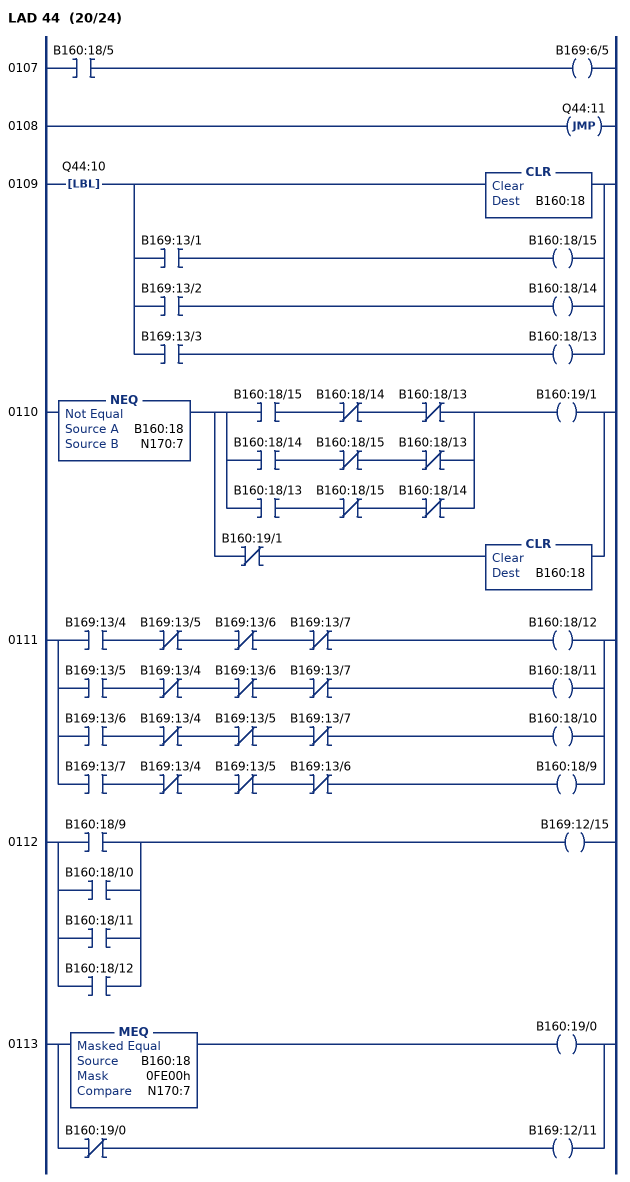
% Rung: 107 %
SOR XIC B160:18/5 OTE B169:6/5 EOR
% Rung: 108 %
SOR JMP Q44:11 EOR
% Rung: 109 %
SOR LBL Q44:10 BST CLR B160:18 NXB XIC B169:13/1 OTE B160:18/15 NXB XIC B169:13/2 OTE B160:18/14 NXB XIC B169:13/3 OTE B160:18/13 BND EOR
% Rung: 110 %
SOR NEQ B160:18 N170:7 BST BST XIC B160:18/15 XIO B160:18/14 XIO B160:18/13 NXB XIC B160:18/14 XIO B160:18/15 XIO B160:18/13 NXB XIC B160:18/13 XIO B160:18/15 XIO B160:18/14 BND OTE B160:19/1 NXB XIO B160:19/1 CLR B160:18 BND EOR
% Rung: 111 %
SOR BST XIC B169:13/4 XIO B169:13/5 XIO B169:13/6 XIO B169:13/7 OTE B160:18/12 NXB XIC B169:13/5 XIO B169:13/4 XIO B169:13/6 XIO B169:13/7 OTE B160:18/11 NXB XIC B169:13/6 XIO B169:13/4 XIO B169:13/5 XIO B169:13/7 OTE B160:18/10 NXB XIC B169:13/7 XIO B169:13/4 XIO B169:13/5 XIO B169:13/6 OTE B160:18/9 BND EOR
% Rung: 112 %
SOR BST XIC B160:18/9 NXB XIC B160:18/10 NXB XIC B160:18/11 NXB XIC B160:18/12 BND OTE B169:12/15 EOR
% Rung: 113 %
SOR BST MEQ B160:18 0FE00h N170:7 OTE B160:19/0 NXB XIO B160:19/0 OTE B169:12/11 BND EOR

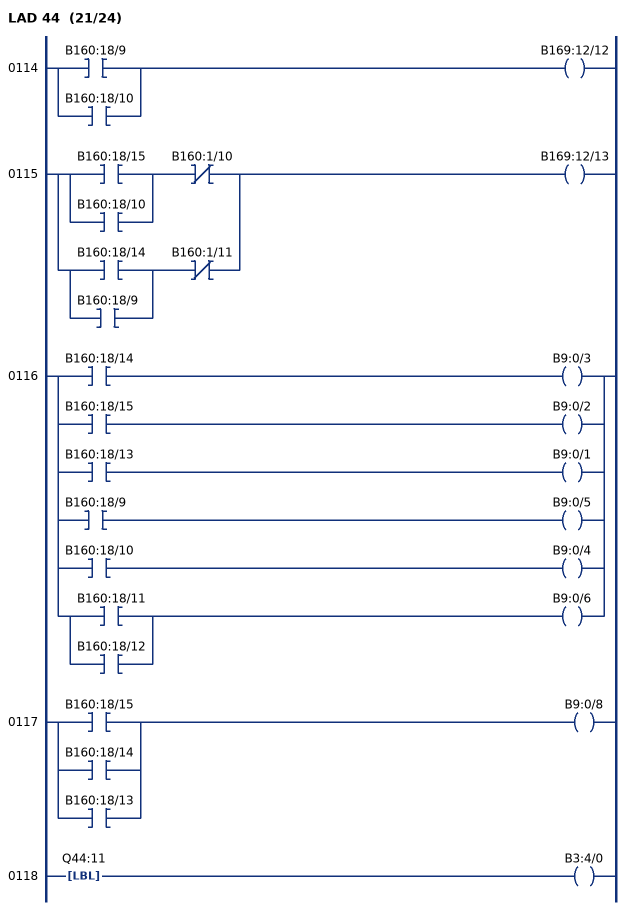
% Rung: 114 %
SOR BST XIC B160:18/9 NXB XIC B160:18/10 BND OTE B169:12/12 EOR
% Rung: 115 %
SOR BST BST XIC B160:18/15 NXB XIC B160:18/10 BND XIO B160:1/10 NXB BST XIC B160:18/14 NXB XIC B160:18/9 BND XIO B160:1/11 BND OTE B169:12/13 EOR
% Rung: 116 %
SOR BST XIC B160:18/14 OTE B9:0/3 NXB XIC B160:18/15 OTE B9:0/2 NXB XIC B160:18/13 OTE B9:0/1 NXB XIC B160:18/9 OTE B9:0/5 NXB XIC B160:18/10 OTE B9:0/4 NXB BST XIC B160:18/11 NXB XIC B160:18/12 BND OTE B9:0/6 BND EOR
% Rung: 117 %
SOR BST XIC B160:18/15 NXB XIC B160:18/14 NXB XIC B160:18/13 BND OTE B9:0/8 EOR
% Rung: 118 %
SOR LBL Q44:11 OTE B3:4/0 EOR

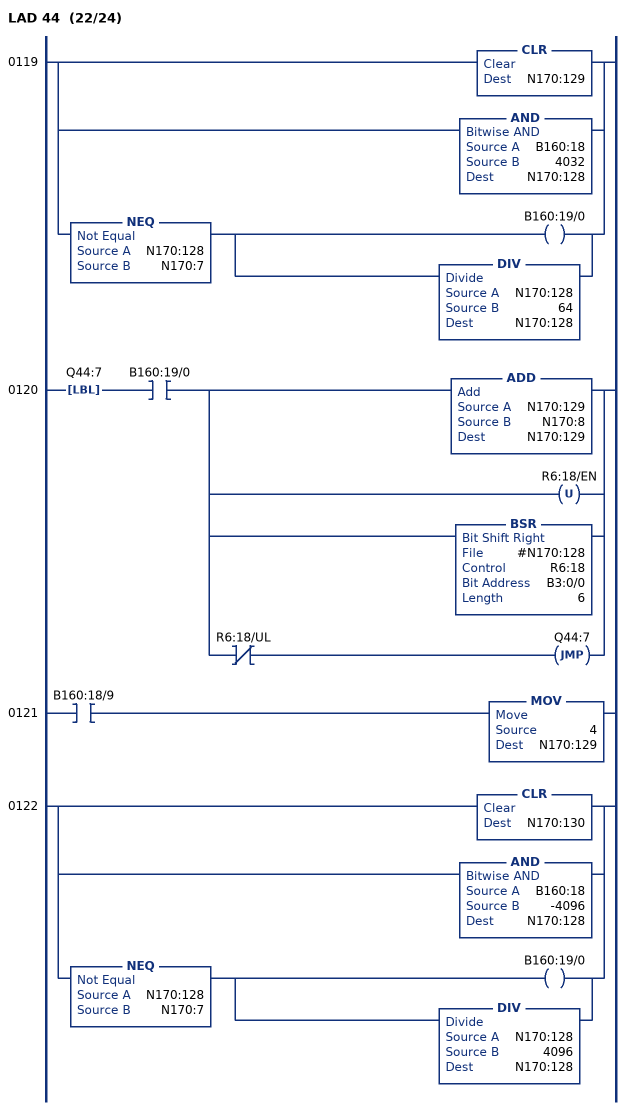
% Rung: 119 %
SOR BST CLR N170:129 NXB AND B160:18 4032 N170:128 NXB NEQ N170:128 N170:7 BST OTE B160:19/0 NXB DIV N170:128 64 N170:128 BND BND EOR
% Rung: 120 %
SOR LBL Q44:7 XIC B160:19/0 BST ADD N170:129 N170:8 N170:129 NXB OTU R6:18/EN NXB BSR #N170:128 R6:18 B3:0/0 6 NXB XIO R6:18/UL JMP Q44:7 BND EOR
% Rung: 121 %
SOR XIC B160:18/9 MOV 4 N170:129 EOR
% Rung: 122 %
SOR BST CLR N170:130 NXB AND B160:18 -4096 N170:128 NXB NEQ N170:128 N170:7 BST OTE B160:19/0 NXB DIV N170:128 4096 N170:128 BND BND EOR

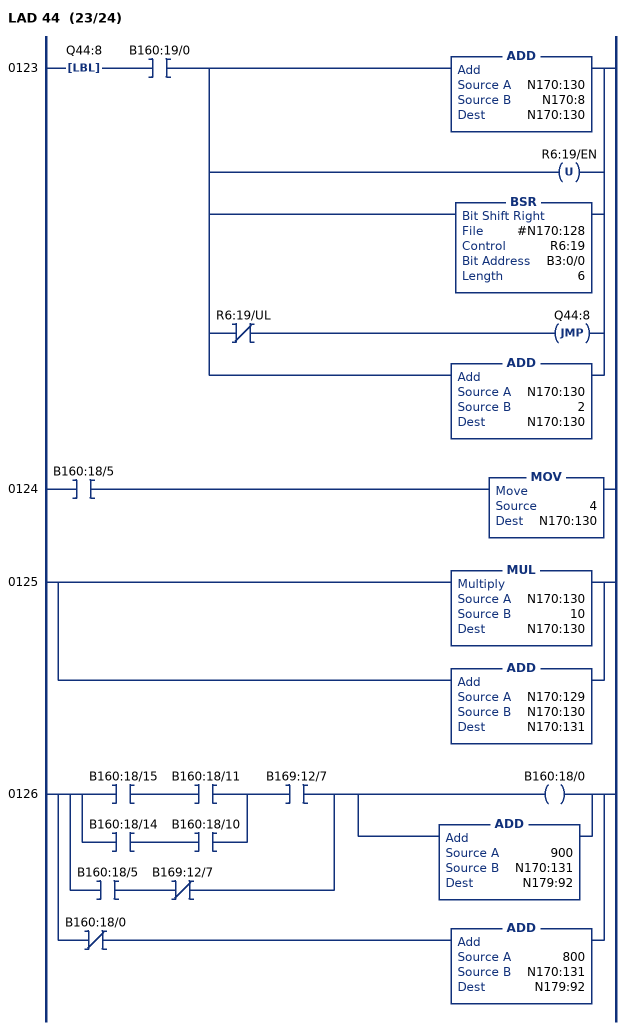
% Rung: 123 %
SOR LBL Q44:8 XIC B160:19/0 BST ADD N170:130 N170:8 N170:130 NXB OTU R6:19/EN NXB BSR #N170:128 R6:19 B3:0/0 6 NXB XIO R6:19/UL JMP Q44:8 NXB ADD N170:130 2 N170:130 BND EOR
% Rung: 124 %
SOR XIC B160:18/5 MOV 4 N170:130 EOR
% Rung: 125 %
SOR BST MUL N170:130 10 N170:130 NXB ADD N170:129 N170:130 N170:131 BND EOR
% Rung: 126 %
SOR BST BST BST XIC B160:18/15 XIC B160:18/11 NXB XIC B160:18/14 XIC B160:18/10 BND XIC B169:12/7 NXB XIC B160:18/5 XIO B169:12/7 BND BST OTE B160:18/0 NXB ADD 900 N170:131 N179:92 BND NXB XIO B160:18/0 ADD 800 N170:131 N179:92 BND EOR

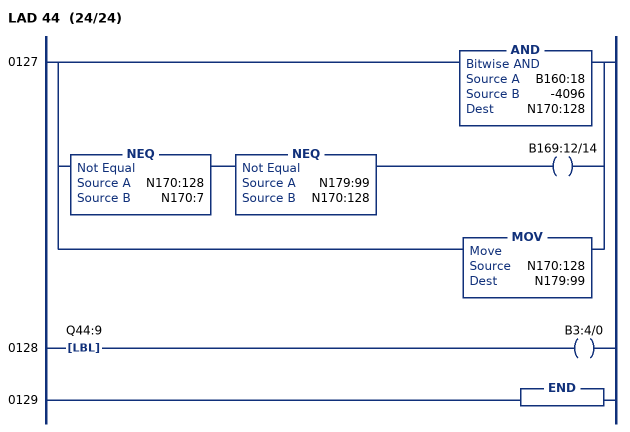
% Rung: 127 %
SOR BST AND B160:18 -4096 N170:128 NXB NEQ N170:128 N170:7 NEQ N179:99 N170:128 OTE B169:12/14 NXB MOV N170:128 N179:99 BND EOR
% Rung: 128 %
SOR LBL Q44:9 OTE B3:4/0 EOR
% Rung: 129 %
SOR END EOR

LADDER 45
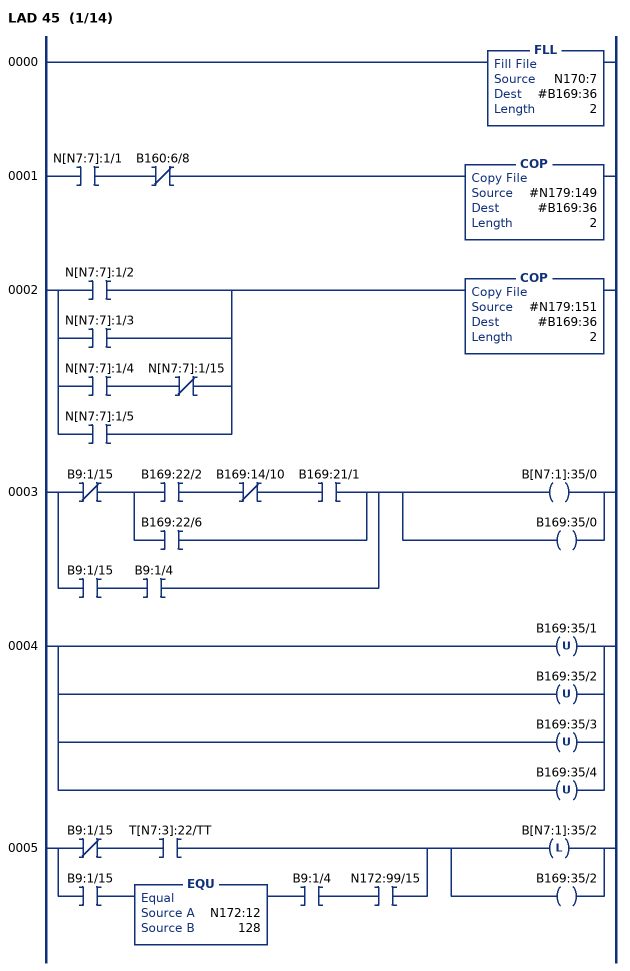
% Rung: 0 %
SOR FLL N170:7 #B169:36 2 EOR
% Rung: 1 %
SOR XIC N[N7:7]:1/1 XIO B160:6/8 COP #N179:149 #B169:36 2 EOR
% Rung: 2 %
SOR BST XIC N[N7:7]:1/2 NXB XIC N[N7:7]:1/3 NXB XIC N[N7:7]:1/4 XIO N[N7:7]:1/15 NXB XIC N[N7:7]:1/5 BND COP #N179:151 #B169:36 2 EOR
% Rung: 3 %
SOR BST XIO B9:1/15 BST XIC B169:22/2 XIO B169:14/10 XIC B169:21/1 NXB XIC B169:22/6 BND NXB XIC B9:1/15 XIC B9:1/4 BND BST OTE B[N7:1]:35/0 NXB OTE B169:35/0 BND EOR
% Rung: 4 %
SOR BST OTU B169:35/1 NXB OTU B169:35/2 NXB OTU B169:35/3 NXB OTU B169:35/4 BND EOR
% Rung: 5 %
SOR BST XIO B9:1/15 XIC T[N7:3]:22/TT NXB XIC B9:1/15 EQU N172:12 128 XIC B9:1/4 XIC N172:99/15 BND BST OTL B[N7:1]:35/2 NXB OTE B169:35/2 BND EOR

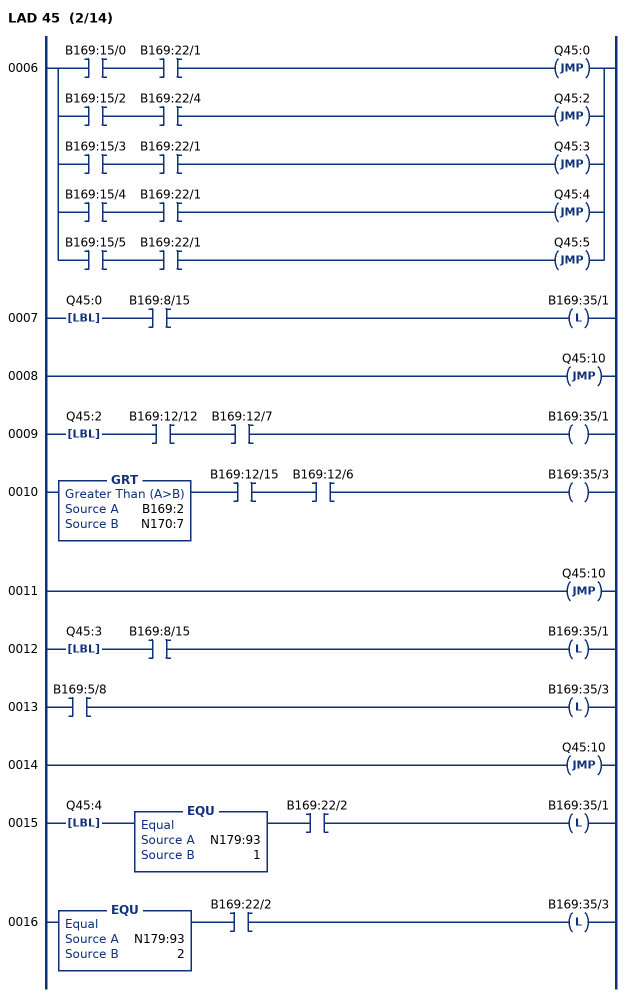
% Rung: 6 %
SOR BST XIC B169:15/0 XIC B169:22/1 JMP Q45:0 NXB XIC B169:15/2 XIC B169:22/4 JMP Q45:2 NXB XIC B169:15/3 XIC B169:22/1 JMP Q45:3 NXB XIC B169:15/4 XIC B169:22/1 JMP Q45:4 NXB XIC B169:15/5 XIC B169:22/1 JMP Q45:5 BND EOR
% Rung: 7 %
SOR LBL Q45:0 XIC B169:8/15 OTL B169:35/1 EOR
% Rung: 8 %
SOR JMP Q45:10 EOR
% Rung: 9 %
SOR LBL Q45:2 XIC B169:12/12 XIC B169:12/7 OTE B169:35/1 EOR
% Rung: 10 %
SOR GRT B169:2 N170:7 XIC B169:12/15 XIC B169:12/6 OTE B169:35/3 EOR
% Rung: 11 %
SOR JMP Q45:10 EOR
% Rung: 12 %
SOR LBL Q45:3 XIC B169:8/15 OTL B169:35/1 EOR
% Rung: 13 %
SOR XIC B169:5/8 OTL B169:35/3 EOR
% Rung: 14 %
SOR JMP Q45:10 EOR
% Rung: 15 %
SOR LBL Q45:4 EQU N179:93 1 XIC B169:22/2 OTL B169:35/1 EOR
% Rung: 16 %
SOR EQU N179:93 2 XIC B169:22/2 OTL B169:35/3 EOR

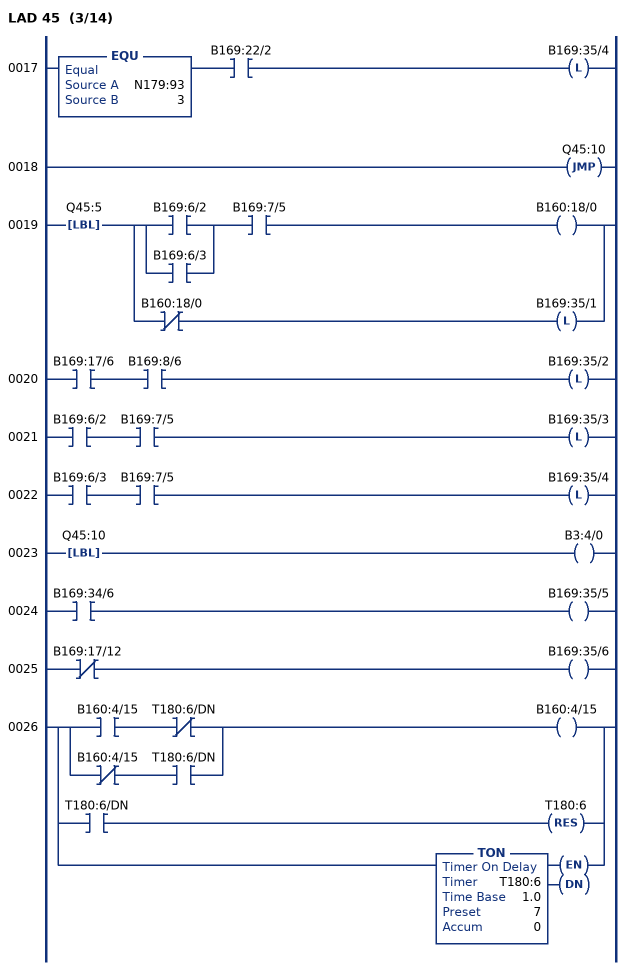
% Rung: 17 %
SOR EQU N179:93 3 XIC B169:22/2 OTL B169:35/4 EOR
% Rung: 18 %
SOR JMP Q45:10 EOR
% Rung: 19 %
SOR LBL Q45:5 BST BST XIC B169:6/2 NXB XIC B169:6/3 BND XIC B169:7/5 OTE B160:18/0 NXB XIO B160:18/0 OTL B169:35/1 BND EOR
% Rung: 20 %
SOR XIC B169:17/6 XIC B169:8/6 OTL B169:35/2 EOR
% Rung: 21 %
SOR XIC B169:6/2 XIC B169:7/5 OTL B169:35/3 EOR
% Rung: 22 %
SOR XIC B169:6/3 XIC B169:7/5 OTL B169:35/4 EOR
% Rung: 23 %
SOR LBL Q45:10 OTE B3:4/0 EOR
% Rung: 24 %
SOR XIC B169:34/6 OTE B169:35/5 EOR
% Rung: 25 %
SOR XIO B169:17/12 OTE B169:35/6 EOR
% Rung: 26 %
SOR BST BST XIC B160:4/15 XIO T180:6/DN NXB XIO B160:4/15 XIC T180:6/DN BND OTE B160:4/15 NXB XIC T180:6/DN RES T180:6 NXB TON T180:6 1.0 7 0 BND EOR

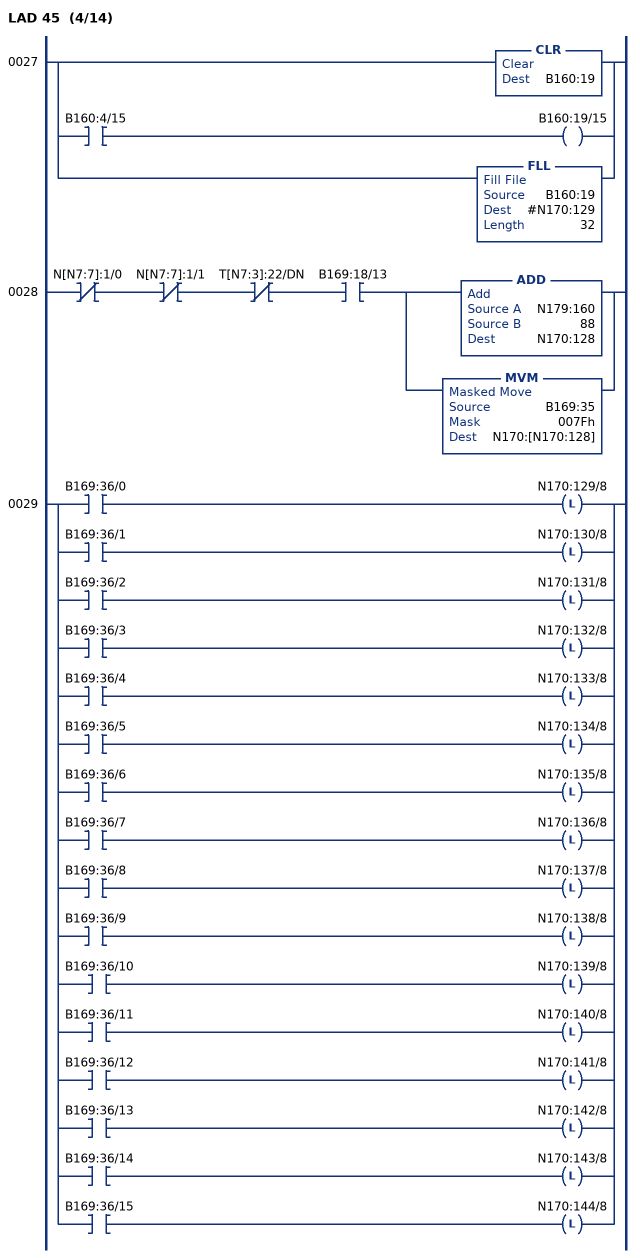
% Rung: 27 %
SOR BST CLR B160:19 NXB XIC B160:4/15 OTE B160:19/15 NXB FLL B160:19 #N170:129 32 BND EOR
% Rung: 28 %
SOR XIO N[N7:7]:1/0 XIO N[N7:7]:1/1 XIO T[N7:3]:22/DN XIC B169:18/13 BST ADD N179:160 88 N170:128 NXB MVM B169:35 007Fh N170:[N170:128] BND EOR
% Rung: 29 %
SOR BST XIC B169:36/0 OTL N170:129/8 NXB XIC B169:36/1 OTL N170:130/8 NXB XIC B169:36/2 OTL N170:131/8 NXB XIC B169:36/3 OTL N170:132/8 NXB XIC B169:36/4 OTL N170:133/8 NXB XIC B169:36/5 OTL N170:134/8 NXB XIC B169:36/6 OTL N170:135/8 NXB XIC B169:36/7 OTL N170:136/8 NXB XIC B169:36/8 OTL N170:137/8 NXB XIC B169:36/9 OTL N170:138/8 NXB XIC B169:36/10 OTL N170:139/8 NXB XIC B169:36/11 OTL N170:140/8 NXB XIC B169:36/12 OTL N170:141/8 NXB XIC B169:36/13 OTL N170:142/8 NXB XIC B169:36/14 OTL N170:143/8 NXB XIC B169:36/15 OTL N170:144/8 BND EOR

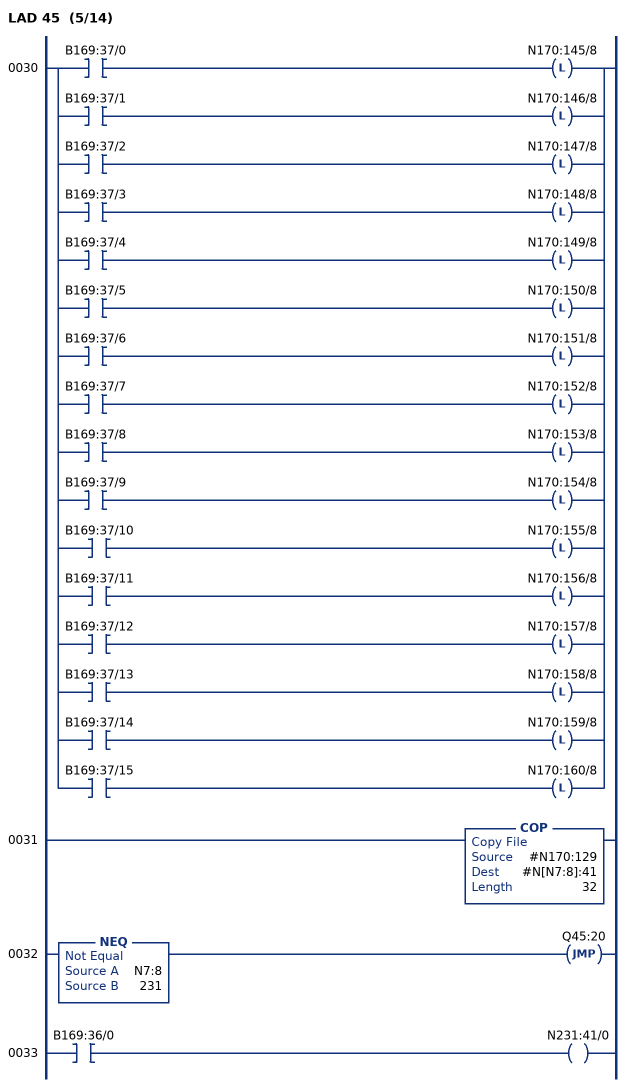
% Rung: 30 %
SOR BST XIC B169:37/0 OTL N170:145/8 NXB XIC B169:37/1 OTL N170:146/8 NXB XIC B169:37/2 OTL N170:147/8 NXB XIC B169:37/3 OTL N170:148/8 NXB XIC B169:37/4 OTL N170:149/8 NXB XIC B169:37/5 OTL N170:150/8 NXB XIC B169:37/6 OTL N170:151/8 NXB XIC B169:37/7 OTL N170:152/8 NXB XIC B169:37/8 OTL N170:153/8 NXB XIC B169:37/9 OTL N170:154/8 NXB XIC B169:37/10 OTL N170:155/8 NXB XIC B169:37/11 OTL N170:156/8 NXB XIC B169:37/12 OTL N170:157/8 NXB XIC B169:37/13 OTL N170:158/8 NXB XIC B169:37/14 OTL N170:159/8 NXB XIC B169:37/15 OTL N170:160/8 BND EOR
% Rung: 31 %
SOR COP #N170:129 #N[N7:8]:41 32 EOR
% Rung: 32 %
SOR NEQ N7:8 231 JMP Q45:20 EOR
% Rung: 33 %
SOR XIC B169:36/0 OTE N231:41/0 EOR

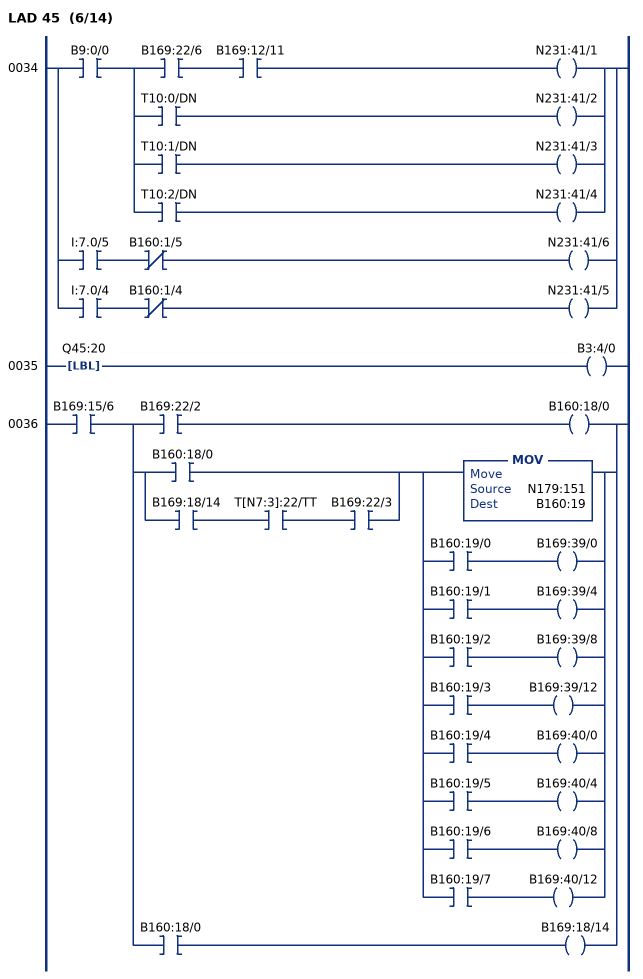
% Rung: 34 %
SOR BST XIC B9:0/0 BST XIC B169:22/6 XIC B169:12/11 OTE N231:41/1 NXB XIC T10:0/DN OTE N231:41/2 NXB XIC T10:1/DN OTE N231:41/3 NXB XIC T10:2/DN OTE N231:41/4 BND NXB XIC I:7.0/5 XIO B160:1/5 OTE N231:41/6 NXB XIC I:7.0/4 XIO B160:1/4 OTE N231:41/5 BND EOR
% Rung: 35 %
SOR LBL Q45:20 OTE B3:4/0 EOR
% Rung: 36 %
SOR XIC B169:15/6 BST XIC B169:22/2 OTE B160:18/0 NXB BST XIC B160:18/0 NXB XIC B169:18/14 XIC T[N7:3]:22/TT XIC B169:22/3 BND BST MOV N179:151 B160:19 NXB XIC B160:19/0 OTE B169:39/0 NXB XIC B160:19/1 OTE B169:39/4 NXB XIC B160:19/2 OTE B169:39/8 NXB XIC B160:19/3 OTE B169:39/12 NXB XIC B160:19/4 OTE B169:40/0 NXB XIC B160:19/5 OTE B169:40/4 NXB XIC B160:19/6 OTE B169:40/8 NXB XIC B160:19/7 OTE B169:40/12 BND NXB XIC B160:18/0 OTE B169:18/14 BND EOR

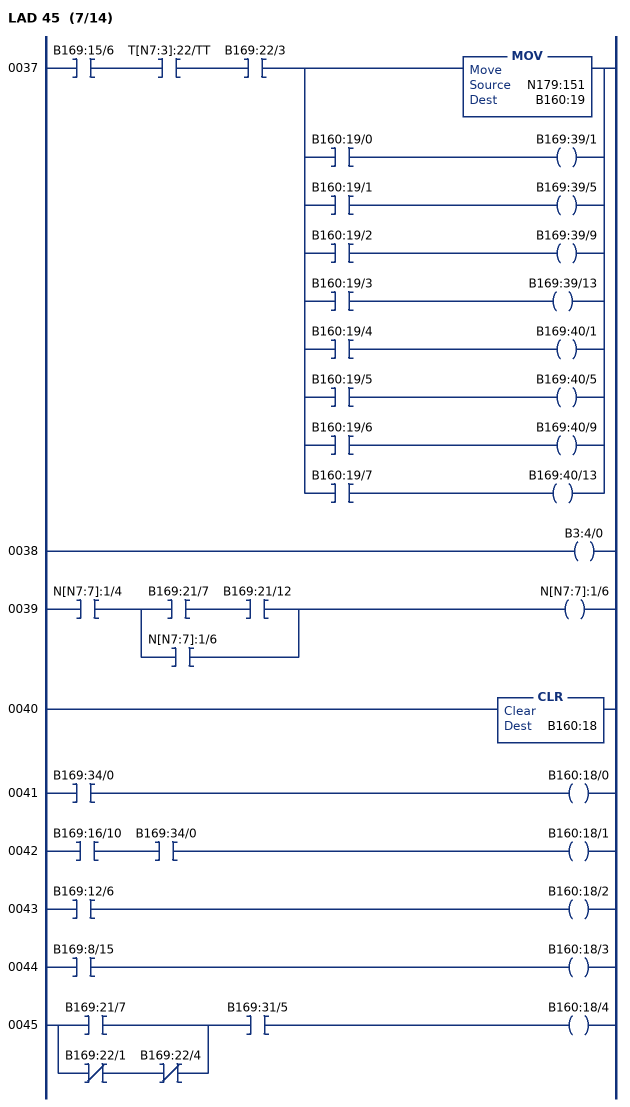
% Rung: 37 %
SOR XIC B169:15/6 XIC T[N7:3]:22/TT XIC B169:22/3 BST MOV N179:151 B160:19 NXB XIC B160:19/0 OTE B169:39/1 NXB XIC B160:19/1 OTE B169:39/5 NXB XIC B160:19/2 OTE B169:39/9 NXB XIC B160:19/3 OTE B169:39/13 NXB XIC B160:19/4 OTE B169:40/1 NXB XIC B160:19/5 OTE B169:40/5 NXB XIC B160:19/6 OTE B169:40/9 NXB XIC B160:19/7 OTE B169:40/13 BND EOR
% Rung: 38 %
SOR OTE B3:4/0 EOR
% Rung: 39 %
SOR XIC N[N7:7]:1/4 BST XIC B169:21/7 XIC B169:21/12 NXB XIC N[N7:7]:1/6 BND OTE N[N7:7]:1/6 EOR
% Rung: 40 %
SOR CLR B160:18 EOR
% Rung: 41 %
SOR XIC B169:34/0 OTE B160:18/0 EOR
% Rung: 42 %
SOR XIC B169:16/10 XIC B169:34/0 OTE B160:18/1 EOR
% Rung: 43 %
SOR XIC B169:12/6 OTE B160:18/2 EOR
% Rung: 44 %
SOR XIC B169:8/15 OTE B160:18/3 EOR
% Rung: 45 %
SOR BST XIC B169:21/7 NXB XIO B169:22/1 XIO B169:22/4 BND XIC B169:31/5 OTE B160:18/4 EOR

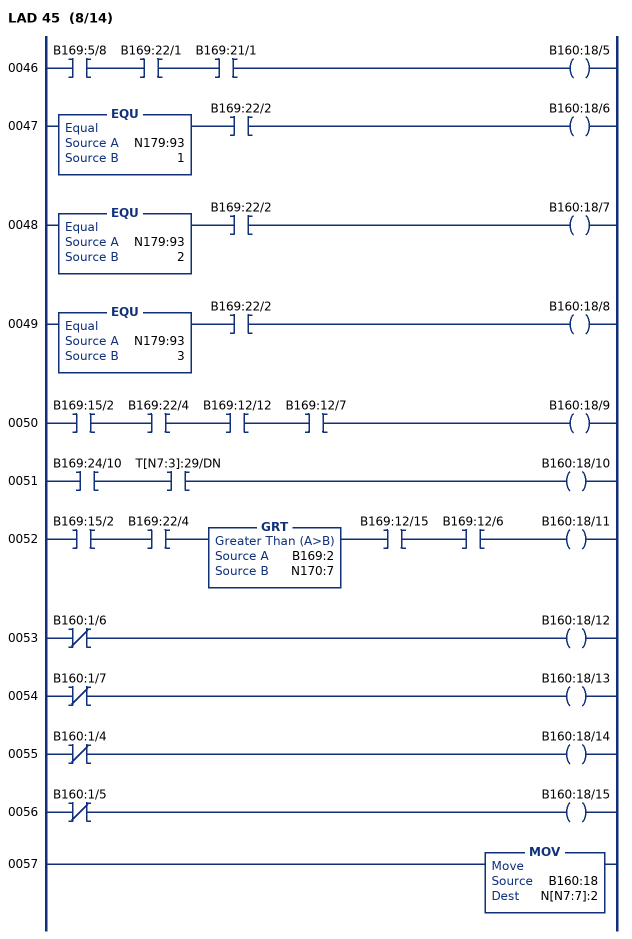
% Rung: 46 %
SOR XIC B169:5/8 XIC B169:22/1 XIC B169:21/1 OTE B160:18/5 EOR
% Rung: 47 %
SOR EQU N179:93 1 XIC B169:22/2 OTE B160:18/6 EOR
% Rung: 48 %
SOR EQU N179:93 2 XIC B169:22/2 OTE B160:18/7 EOR
% Rung: 49 %
SOR EQU N179:93 3 XIC B169:22/2 OTE B160:18/8 EOR
% Rung: 50 %
SOR XIC B169:15/2 XIC B169:22/4 XIC B169:12/12 XIC B169:12/7 OTE B160:18/9 EOR
% Rung: 51 %
SOR XIC B169:24/10 XIC T[N7:3]:29/DN OTE B160:18/10 EOR
% Rung: 52 %
SOR XIC B169:15/2 XIC B169:22/4 GRT B169:2 N170:7 XIC B169:12/15 XIC B169:12/6 OTE B160:18/11 EOR
% Rung: 53 %
SOR XIO B160:1/6 OTE B160:18/12 EOR
% Rung: 54 %
SOR XIO B160:1/7 OTE B160:18/13 EOR
% Rung: 55 %
SOR XIO B160:1/4 OTE B160:18/14 EOR
% Rung: 56 %
SOR XIO B160:1/5 OTE B160:18/15 EOR
% Rung: 57 %
SOR MOV B160:18 N[N7:7]:2 EOR

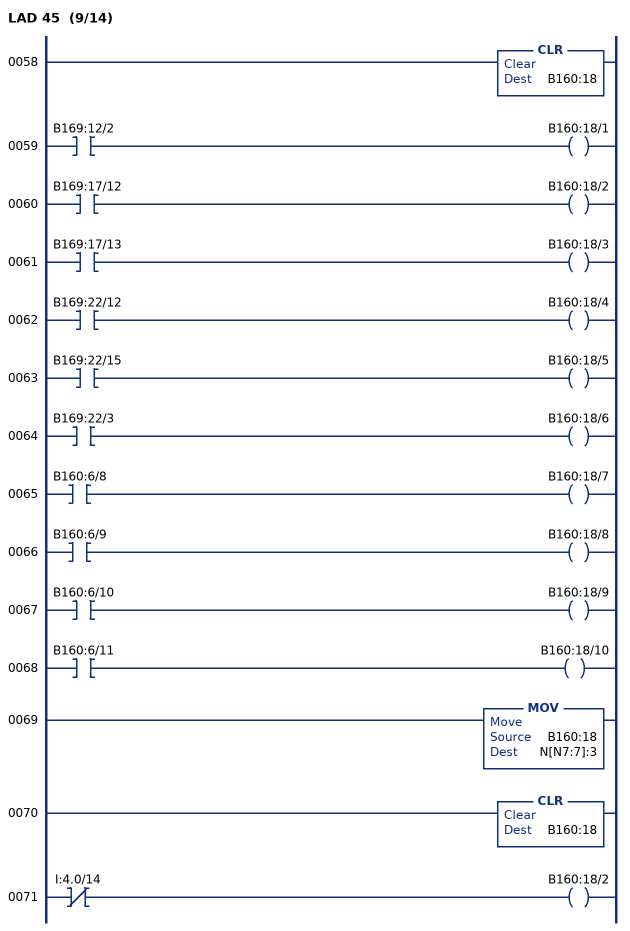
% Rung: 58 %
SOR CLR B160:18 EOR
% Rung: 59 %
SOR XIC B169:12/2 OTE B160:18/1 EOR
% Rung: 60 %
SOR XIC B169:17/12 OTE B160:18/2 EOR
% Rung: 61 %
SOR XIC B169:17/13 OTE B160:18/3 EOR
% Rung: 62 %
SOR XIC B169:22/12 OTE B160:18/4 EOR
% Rung: 63 %
SOR XIC B169:22/15 OTE B160:18/5 EOR
% Rung: 64 %
SOR XIC B169:22/3 OTE B160:18/6 EOR
% Rung: 65 %
SOR XIC B160:6/8 OTE B160:18/7 EOR
% Rung: 66 %
SOR XIC B160:6/9 OTE B160:18/8 EOR
% Rung: 67 %
SOR XIC B160:6/10 OTE B160:18/9 EOR
% Rung: 68 %
SOR XIC B160:6/11 OTE B160:18/10 EOR
% Rung: 69 %
SOR MOV B160:18 N[N7:7]:3 EOR
% Rung: 70 %
SOR CLR B160:18 EOR
% Rung: 71 %
SOR XIO I:4.0/14 OTE B160:18/2 EOR

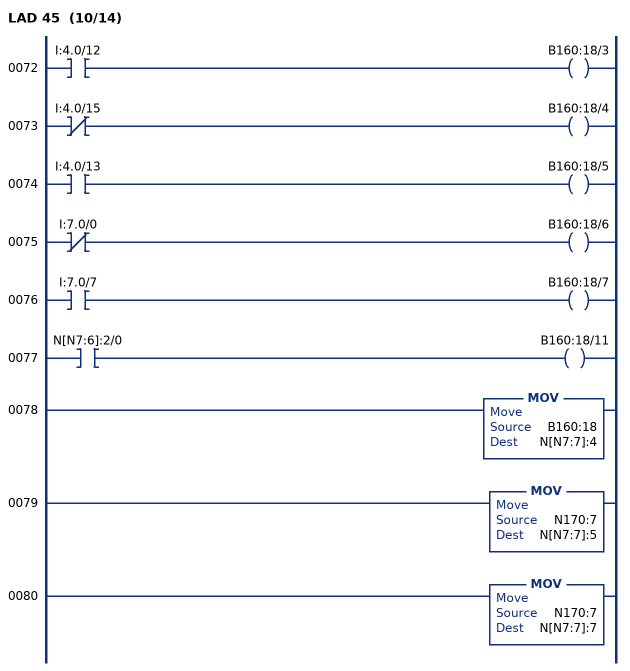
% Rung: 72 %
SOR XIC I:4.0/12 OTE B160:18/3 EOR
% Rung: 73 %
SOR XIO I:4.0/15 OTE B160:18/4 EOR
% Rung: 74 %
SOR XIC I:4.0/13 OTE B160:18/5 EOR
% Rung: 75 %
SOR XIO I:7.0/0 OTE B160:18/6 EOR
% Rung: 76 %
SOR XIC I:7.0/7 OTE B160:18/7 EOR
% Rung: 77 %
SOR XIC N[N7:6]:2/0 OTE B160:18/11 EOR
% Rung: 78 %
SOR MOV B160:18 N[N7:7]:4 EOR
% Rung: 79 %
SOR MOV N170:7 N[N7:7]:5 EOR
% Rung: 80 %
SOR MOV N170:7 N[N7:7]:7 EOR

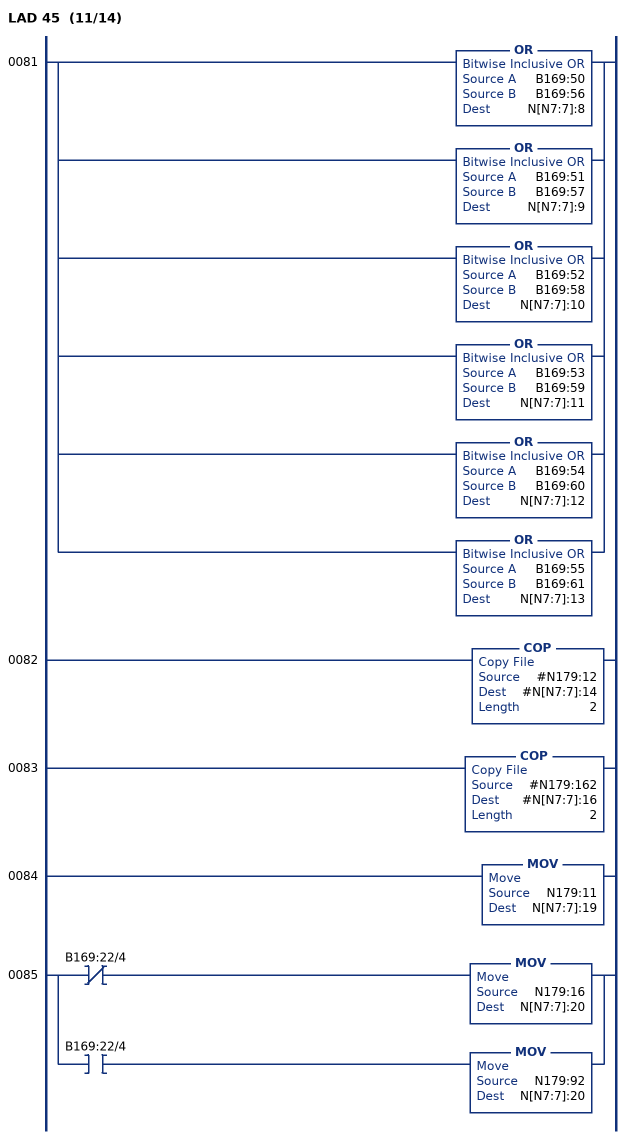
% Rung: 81 %
SOR BST OR B169:50 B169:56 N[N7:7]:8 NXB OR B169:51 B169:57 N[N7:7]:9 NXB OR B169:52 B169:58 N[N7:7]:10 NXB OR B169:53 B169:59 N[N7:7]:11 NXB OR B169:54 B169:60 N[N7:7]:12 NXB OR B169:55 B169:61 N[N7:7]:13 BND EOR
% Rung: 82 %
SOR COP #N179:12 #N[N7:7]:14 2 EOR
% Rung: 83 %
SOR COP #N179:162 #N[N7:7]:16 2 EOR
% Rung: 84 %
SOR MOV N179:11 N[N7:7]:19 EOR
% Rung: 85 %
SOR BST XIO B169:22/4 MOV N179:16 N[N7:7]:20 NXB XIC B169:22/4 MOV N179:92 N[N7:7]:20 BND EOR

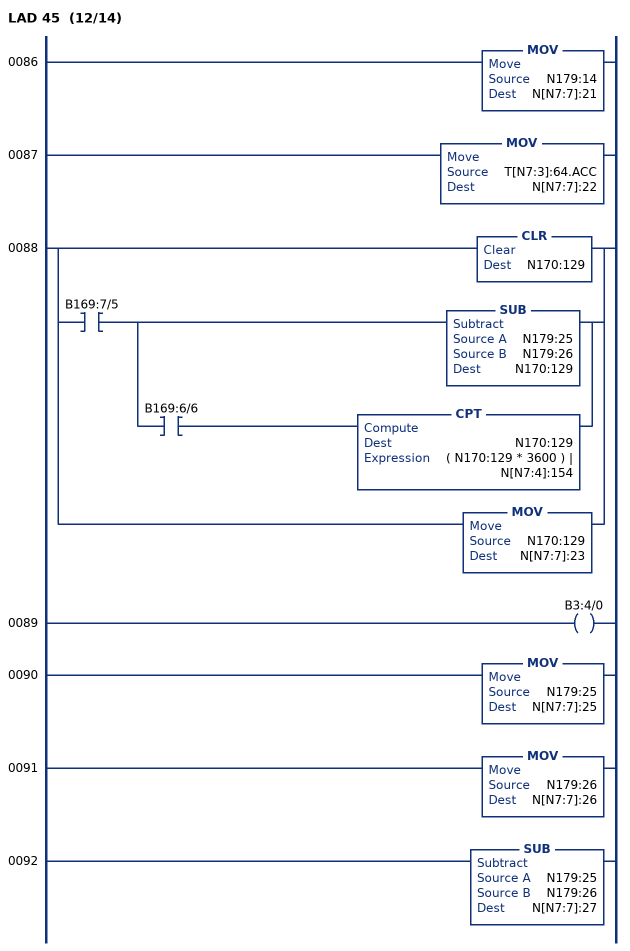
% Rung: 86 %
SOR MOV N179:14 N[N7:7]:21 EOR
% Rung: 87 %
SOR MOV T[N7:3]:64.ACC N[N7:7]:22 EOR
% Rung: 88 %
SOR BST CLR N170:129 NXB XIC B169:7/5 BST SUB N179:25 N179:26 N170:129 NXB XIC B169:6/6 CPT N170:129 " ( N170:129 * 3600 ) | N[N7:4]:154 " BND NXB MOV N170:129 N[N7:7]:23 BND EOR
% Rung: 89 %
SOR OTE B3:4/0 EOR
% Rung: 90 %
SOR MOV N179:25 N[N7:7]:25 EOR
% Rung: 91 %
SOR MOV N179:26 N[N7:7]:26 EOR
% Rung: 92 %
SOR SUB N179:25 N179:26 N[N7:7]:27 EOR

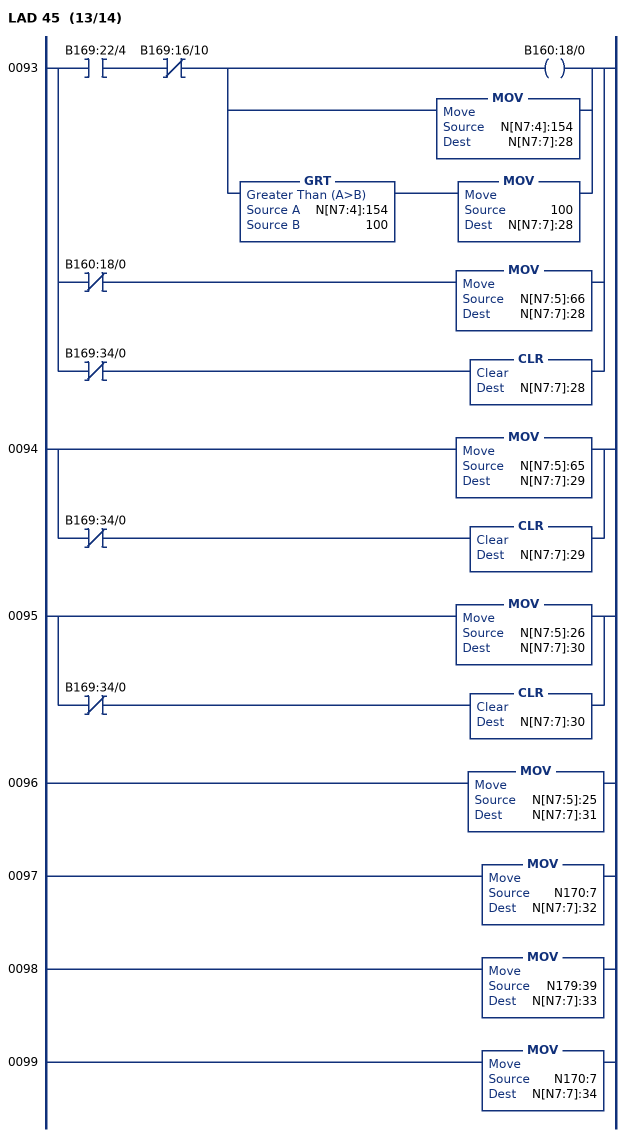
% Rung: 93 %
SOR BST XIC B169:22/4 XIO B169:16/10 BST OTE B160:18/0 NXB MOV N[N7:4]:154 N[N7:7]:28 NXB GRT N[N7:4]:154 100 MOV 100 N[N7:7]:28 BND NXB XIO B160:18/0 MOV N[N7:5]:66 N[N7:7]:28 NXB XIO B169:34/0 CLR N[N7:7]:28 BND EOR
% Rung: 94 %
SOR BST MOV N[N7:5]:65 N[N7:7]:29 NXB XIO B169:34/0 CLR N[N7:7]:29 BND EOR
% Rung: 95 %
SOR BST MOV N[N7:5]:26 N[N7:7]:30 NXB XIO B169:34/0 CLR N[N7:7]:30 BND EOR
% Rung: 96 %
SOR MOV N[N7:5]:25 N[N7:7]:31 EOR
% Rung: 97 %
SOR MOV N170:7 N[N7:7]:32 EOR
% Rung: 98 %
SOR MOV N179:39 N[N7:7]:33 EOR
% Rung: 99 %
SOR MOV N170:7 N[N7:7]:34 EOR

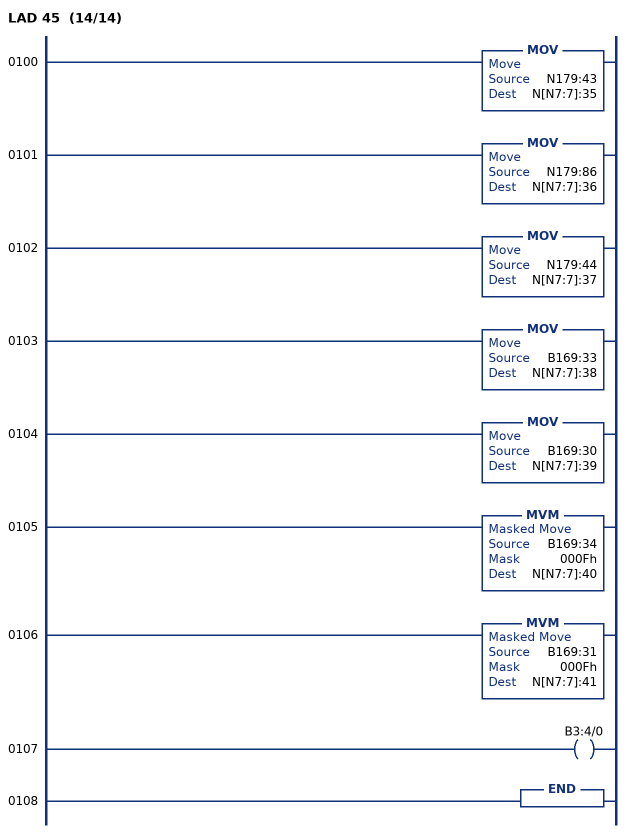
% Rung: 100 %
SOR MOV N179:43 N[N7:7]:35 EOR
% Rung: 101 %
SOR MOV N179:86 N[N7:7]:36 EOR
% Rung: 102 %
SOR MOV N179:44 N[N7:7]:37 EOR
% Rung: 103 %
SOR MOV B169:33 N[N7:7]:38 EOR
% Rung: 104 %
SOR MOV B169:30 N[N7:7]:39 EOR
% Rung: 105 %
SOR MVM B169:34 000Fh N[N7:7]:40 EOR
% Rung: 106 %
SOR MVM B169:31 000Fh N[N7:7]:41 EOR
% Rung: 107 %
SOR OTE B3:4/0 EOR
% Rung: 108 %
SOR END EOR

LADDER 50
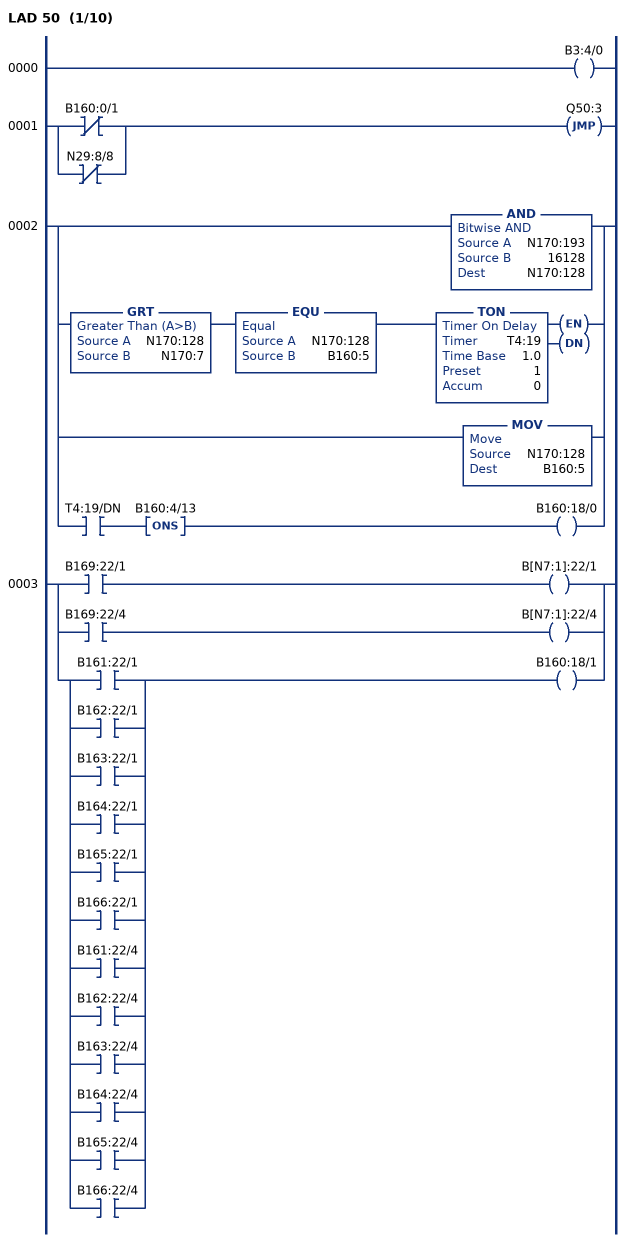
% Rung: 0 %
SOR OTE B3:4/0 EOR
% Rung: 1 %
SOR BST XIO B160:0/1 NXB XIO N29:8/8 BND JMP Q50:3 EOR
% Rung: 2 %
SOR BST AND N170:193 16128 N170:128 NXB GRT N170:128 N170:7 EQU N170:128 B160:5 TON T4:19 1.0 1 0 NXB MOV N170:128 B160:5 NXB XIC T4:19/DN OSR B160:4/13 OTE B160:18/0 BND EOR
% Rung: 3 %
SOR BST XIC B169:22/1 OTE B[N7:1]:22/1 NXB XIC B169:22/4 OTE B[N7:1]:22/4 NXB BST XIC B161:22/1 NXB XIC B162:22/1 NXB XIC B163:22/1 NXB XIC B164:22/1 NXB XIC B165:22/1 NXB XIC B166:22/1 NXB XIC B161:22/4 NXB XIC B162:22/4 NXB XIC B163:22/4 NXB XIC B164:22/4 NXB XIC B165:22/4 NXB XIC B166:22/4 BND OTE B160:18/1 BND EOR

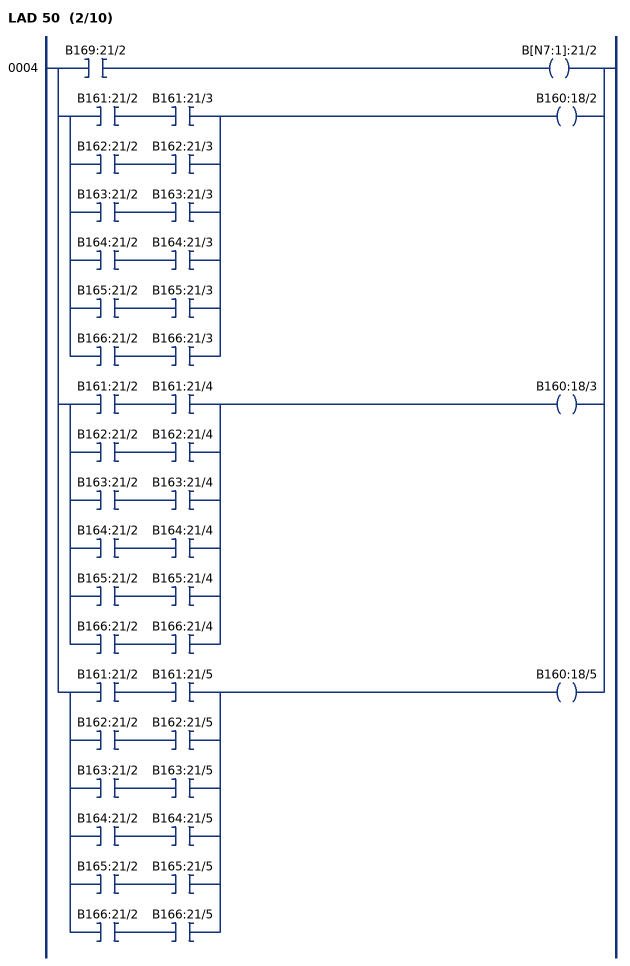
% Rung: 4 %
SOR BST XIC B169:21/2 OTE B[N7:1]:21/2 NXB BST XIC B161:21/2 XIC B161:21/3 NXB XIC B162:21/2 XIC B162:21/3 NXB XIC B163:21/2 XIC B163:21/3 NXB XIC B164:21/2 XIC B164:21/3 NXB XIC B165:21/2 XIC B165:21/3 NXB XIC B166:21/2 XIC B166:21/3 BND OTE B160:18/2 NXB BST XIC B161:21/2 XIC B161:21/4 NXB XIC B162:21/2 XIC B162:21/4 NXB XIC B163:21/2 XIC B163:21/4 NXB XIC B164:21/2 XIC B164:21/4 NXB XIC B165:21/2 XIC B165:21/4 NXB XIC B166:21/2 XIC B166:21/4 BND OTE B160:18/3 NXB BST XIC B161:21/2 XIC B161:21/5 NXB XIC B162:21/2 XIC B162:21/5 NXB XIC B163:21/2 XIC B163:21/5 NXB XIC B164:21/2 XIC B164:21/5 NXB XIC B165:21/2 XIC B165:21/5 NXB XIC B166:21/2 XIC B166:21/5 BND OTE B160:18/5 BND EOR

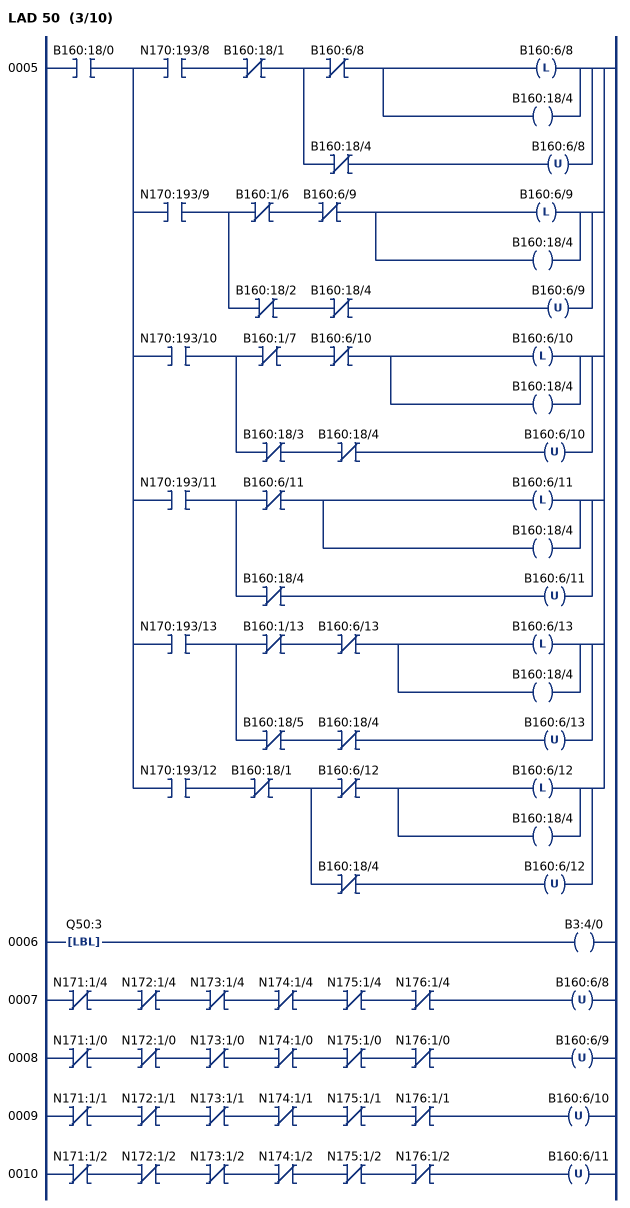
% Rung: 5 %
SOR XIC B160:18/0 BST XIC N170:193/8 XIO B160:18/1 BST XIO B160:6/8 BST OTL B160:6/8 NXB OTE B160:18/4 BND NXB XIO B160:18/4 OTU B160:6/8 BND NXB XIC N170:193/9 BST XIO B160:1/6 XIO B160:6/9 BST OTL B160:6/9 NXB OTE B160:18/4 BND NXB XIO B160:18/2 XIO B160:18/4 OTU B160:6/9 BND NXB XIC N170:193/10 BST XIO B160:1/7 XIO B160:6/10 BST OTL B160:6/10 NXB OTE B160:18/4 BND NXB XIO B160:18/3 XIO B160:18/4 OTU B160:6/10 BND NXB XIC N170:193/11 BST XIO B160:6/11 BST OTL B160:6/11 NXB OTE B160:18/4 BND NXB XIO B160:18/4 OTU B160:6/11 BND NXB XIC N170:193/13 BST XIO B160:1/13 XIO B160:6/13 BST OTL B160:6/13 NXB OTE B160:18/4 BND NXB XIO B160:18/5 XIO B160:18/4 OTU B160:6/13 BND NXB XIC N170:193/12 XIO B160:18/1 BST XIO B160:6/12 BST OTL B160:6/12 NXB OTE B160:18/4 BND NXB XIO B160:18/4 OTU B160:6/12 BND BND EOR
% Rung: 6 %
SOR LBL Q50:3 OTE B3:4/0 EOR
% Rung: 7 %
SOR XIO N171:1/4 XIO N172:1/4 XIO N173:1/4 XIO N174:1/4 XIO N175:1/4 XIO N176:1/4 OTU B160:6/8 EOR
% Rung: 8 %
SOR XIO N171:1/0 XIO N172:1/0 XIO N173:1/0 XIO N174:1/0 XIO N175:1/0 XIO N176:1/0 OTU B160:6/9 EOR
% Rung: 9 %
SOR XIO N171:1/1 XIO N172:1/1 XIO N173:1/1 XIO N174:1/1 XIO N175:1/1 XIO N176:1/1 OTU B160:6/10 EOR
% Rung: 10 %
SOR XIO N171:1/2 XIO N172:1/2 XIO N173:1/2 XIO N174:1/2 XIO N175:1/2 XIO N176:1/2 OTU B160:6/11 EOR

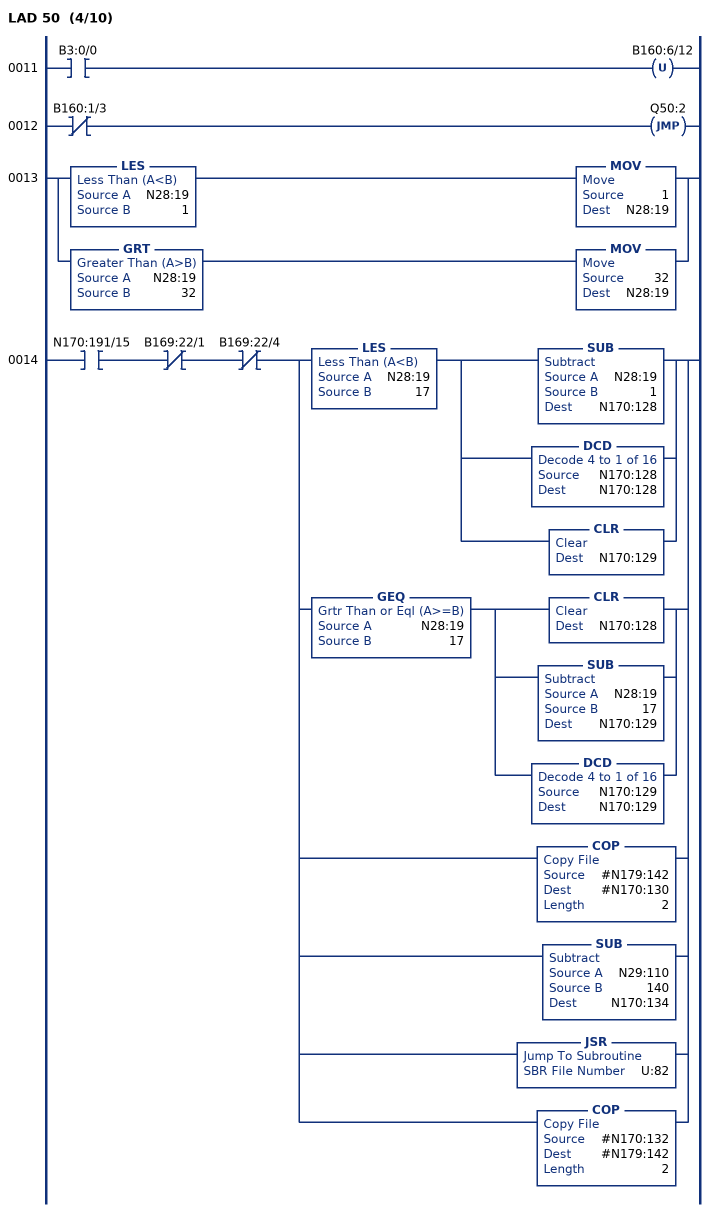
% Rung: 11 %
SOR XIC B3:0/0 OTU B160:6/12 EOR
% Rung: 12 %
SOR XIO B160:1/3 JMP Q50:2 EOR
% Rung: 13 %
SOR BST LES N28:19 1 MOV 1 N28:19 NXB GRT N28:19 32 MOV 32 N28:19 BND EOR
% Rung: 14 %
SOR XIC N170:191/15 XIO B169:22/1 XIO B169:22/4 BST LES N28:19 17 BST SUB N28:19 1 N170:128 NXB DCD N170:128 N170:128 NXB CLR N170:129 BND NXB GEQ N28:19 17 BST CLR N170:128 NXB SUB N28:19 17 N170:129 NXB DCD N170:129 N170:129 BND NXB COP #N179:142 #N170:130 2 NXB SUB N29:110 140 N170:134 NXB JSR U:82 NXB COP #N170:132 #N179:142 2 BND EOR

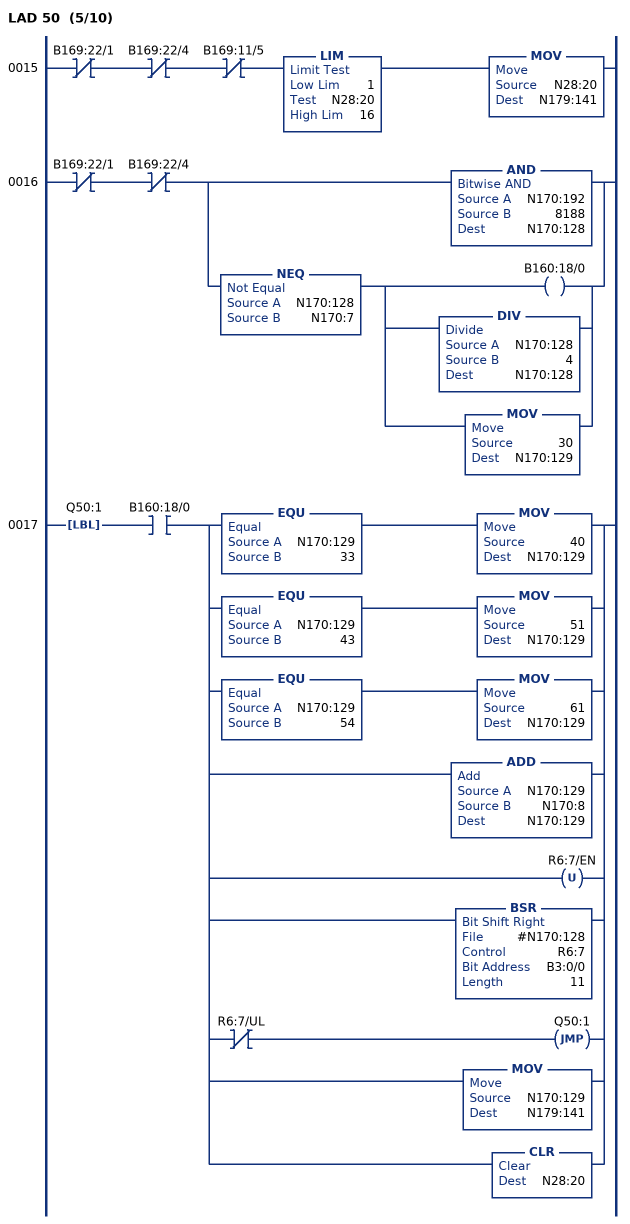
% Rung: 15 %
SOR XIO B169:22/1 XIO B169:22/4 XIO B169:11/5 LIM 1 N28:20 16 MOV N28:20 N179:141 EOR
% Rung: 16 %
SOR XIO B169:22/1 XIO B169:22/4 BST AND N170:192 8188 N170:128 NXB NEQ N170:128 N170:7 BST OTE B160:18/0 NXB DIV N170:128 4 N170:128 NXB MOV 30 N170:129 BND BND EOR
% Rung: 17 %
SOR LBL Q50:1 XIC B160:18/0 BST BST EQU N170:129 33 MOV 40 N170:129 NXB EQU N170:129 43 MOV 51 N170:129 NXB EQU N170:129 54 MOV 61 N170:129 NXB ADD N170:129 N170:8 N170:129 BND NXB OTU R6:7/EN NXB BSR #N170:128 R6:7 B3:0/0 11 NXB XIO R6:7/UL JMP Q50:1 NXB MOV N170:129 N179:141 NXB CLR N28:20 BND EOR

